DATA_BLOCK "PreAlarm_DB"
{ S7_Optimized_Access := 'FALSE' }
VERSION : 0.1
NON_RETAIN
   VAR
      Ana_PreAlarm : Array[1..40] of "UDT_Ana_PreAlarm";   // 模拟量预警信息数组[1..40]
   END_VAR


BEGIN
END_DATA_BLOCK